PROGRAM PRG_HV_ILK
VAR
	HV_ILK_OK: bool := false;
END_VAR


//evaluate the HV ILK_OK bit
//HV_ILK_OK := GCC_40.IG.xAT_VAC;

hv1(i_xExtIlkOK := HV_ILK_OK);
hv2(i_xExtIlkOK := HV_ILK_OK);

END_PROGRAM

(* stored: Version 1.1.0.1, ProductVersion 3.1.4022.12
   POU PRG_HV_ILK: Id {74363be8-caf7-4d2d-8709-16ae5ee5e8a6}, SpecialFunc None *)
